Xinje XDPPro project, PLC1: XD3-16 (software 3.7.18_en 2025-06-04)

PROGRAM Ladder

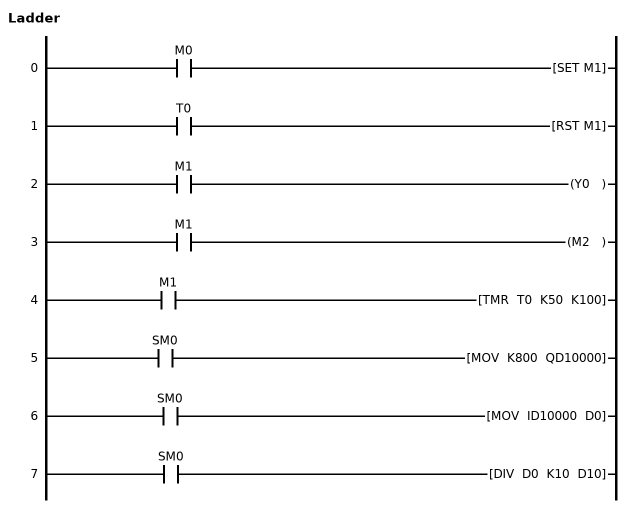
LD     M0
SET    M1
LD     T0
RST    M1
LD     M1
OUT    Y0
LD     M1
OUT    M2
LD     M1
TMR    T0 K50 K100
LD     SM0
MOV    K800 QD10000
LD     SM0
MOV    ID10000 D0
LD     SM0
DIV    D0 K10 D10